// TIA Portal V19 export
FUNCTION "A01_HMI_CALL" : Void   // FC226, LAD
// stored: SetENOAutomatically false
BEGIN

REGION Network 1
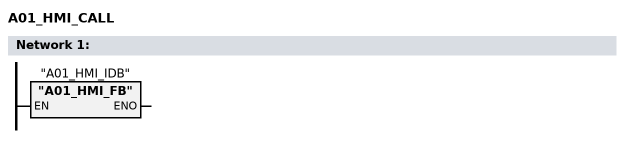
   RUNG wire#powerrail
      "A01_HMI_IDB"()
   END_RUNG
   // the same network as SCL:
   "A01_HMI_IDB"();   // "A01_HMI_FB"
END_REGION
END_FUNCTION
